(* PLC project PlcMain, Beckhoff Automation GmbH TwinCAT PLC Control 3.5.13.21 *)
(* stored: creationDateTime 2022-08-19T12:35:15.5548901, modificationDateTime 2022-08-19T12:35:15.5548901 *)

{attribute 'qualified_only'}
{attribute 'strict'}
TYPE StateHeat :
(
	Off,
	Init,
	Ready,
	Heat,
	Hold,
	Done
);
END_TYPE
